Universal Robots PolyScope program: 4_wash_hover.urp

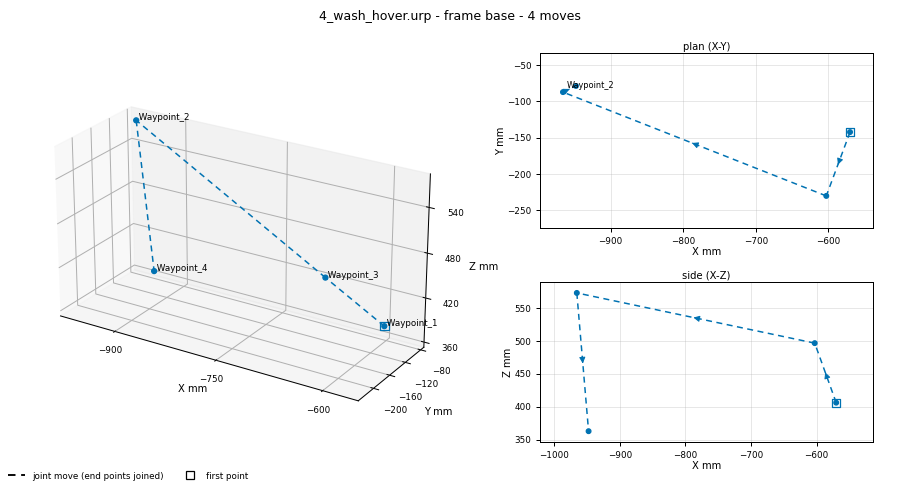
[picture p0: tool path of 4_wash_hover.urp in frame base, 4 of 4 moves have a stored position in this frame; points joined in program order, loops and branches not executed]
Program 4_wash_hover (installation=default directory=/programs/washer_rahman createdIn=5.9.5.1031259 lastSavedIn=5.9.5.1031259 robotSerialNumber=20215500597)
Calibrated DH parameters: a=[0.000193, -0.066673, -0.391568, -0.000012, 0.00005, 0]; d=[0.162643, -472.05677, 465.132521, 7.058239, 0.099746, 0.099582]; alpha=[1.571116, 0.00089, 0.003862, 1.569269, -1.569248, 0]; deltaTheta=[0, -1.413394, 7.628392, 0.068187, 0, -0.000001]
Robot Program (runOnlyOnce=true)
  SuppressedNode
    var_2 := 2
  SuppressedNode
    Script: glass_hover=p[-.603,-0.23+var_2*0.150 ,0.277,2.067,2.652,-2.043]
  SuppressedNode
    Script: glass_hover=p[-.603,-0.23+GP_int_in[0]*0.150 ,0.277,2.067,2.652,-2.043]
  MoveJ speed 60 deg/s, acceleration 80 deg/s^2 (useActiveTCP=true) feature=Base
    Waypoint Waypoint_1: TCP in base x=-570.322 y=-142.143 z=406.231 mm, rx=-1.2552 ry=-1.3745 rz=1.0423 rad; joints [2.423, -96.242, 131.838, -205.844, -93.335, -5.251] deg; TCP offset x=0 y=0 z=191.5 mm, rx=0 ry=0 rz=0 rad
    SuppressedNode
      Waypoint Waypoint (Variable): variable=glass_hover
    Waypoint Waypoint_3: TCP in base x=-603.007 y=-230.009 z=496.953 mm, rx=-1.234 ry=-1.5833 rz=1.2196 rad; joints [5.326, -97.862, 114.523, -182.414, -82.368, -2.596] deg
    SuppressedNode
      Waypoint Waypoint (Variable): variable=wash_hover
    Waypoint Waypoint_2: TCP in base x=-965.488 y=-87.111 z=573.443 mm, rx=-1.3367 ry=-1.4136 rz=1.0288 rad; joints [-3.617, -51.899, 44.548, -158.561, -87.146, -4.428] deg
  MoveL speed 250 mm/s, acceleration 1200 mm/s^2 (useActiveTCP=true) feature=Base
    MoveDirectionNode (selectedDirection=ZMinus)
      Until DISTANCE (allowActions=false deceleration=3 distanceNodeType=STOP) Distance=0.15; motionParameters(blendRadius=0)
  MoveJ speed 60 deg/s, acceleration 80 deg/s^2 (useActiveTCP=true) feature=Base
    Waypoint Waypoint_4: TCP in base x=-947.566 y=-78.667 z=362.787 mm, rx=-1.3565 ry=-1.437 rz=0.8682 rad; joints [-2.082, -50.772, 70.995, -182.432, -94.11, -8.124] deg
